TYPE T_FSS_RejecCode : STRING(40);
END_TYPE

(* stored: Version 1.1.0.1
   DUT T_FSS_RejecCode: Id {5e96b671-8d6d-4355-a9d0-3693119cdf3b} *)
